FUNCTION_BLOCK VolumePump
VAR
	pump						: Relay;
	eState						: ( RESET, START );
	fPumpedJuiceInMililiters	: REAL;
END_VAR

CASE eState OF
	
	RESET:
		pump.SwitchOff();
		fPumpedJuiceInMililiters := 0;
		
	START:
		pump.SwitchOn();
		fPumpedJuiceInMililiters := fPumpedJuiceInMililiters + 10;
		
END_CASE

PROPERTY IsPumping : BOOL
GET
IsPumping := pump.State;
END_GET
END_PROPERTY

PROPERTY PumpedJuiceInMililiters : REAL
GET
PumpedJuiceInMililiters := fPumpedJuiceInMililiters;
END_GET
END_PROPERTY

METHOD Reset : BOOL
VAR_INPUT
END_VAR
eState := RESET;
END_METHOD

METHOD Start : BOOL
VAR_INPUT
END_VAR
eState := START;
END_METHOD

END_FUNCTION_BLOCK

(* stored: Version 1.1.0.1
   POU VolumePump: Id {f0a7faee-552d-4aa6-b633-5280f4c5f76f}, SpecialFunc None
   Property IsPumping: Id {945d2fef-a9ee-4910-b578-d8558166eb0b}
   Get Get: Id {7a6066f1-3e65-4e99-a393-19de9e0eae3a}
   Property PumpedJuiceInMililiters: Id {697b894b-ea98-4121-8d4f-72ecccba8c42}
   Get Get: Id {2441b756-a90f-456a-96f6-1dc737a393aa}
   Method Reset: Id {fae4d1d0-68cf-4747-9897-b0426c8c086b}
   Method Start: Id {74a2eead-d63f-4aaa-8c08-33ad3a461f4d} *)
